(* PLC project Wiimote example, Beremiz Beremiz 1 *)
(* stored: creationDateTime 2012-09-12T23:30:19, modificationDateTime 2017-06-06T13:10:31 *)

PROGRAM main
  VAR
    x : INT;
    y : INT;
    a : INT;
    b : INT;
    c : INT;
    b1 : WORD;
    b0 : WORD;
  END_VAR
  VAR_EXTERNAL
    WiiNunchuckStickX : INT;
    WiiNunchuckStickY : INT;
    WiiNunchuckButtons : WORD;
    WiiButtons : WORD;
    WiiNunchuckAccX : INT;
    WiiNunchuckAccY : INT;
    WiiNunchuckAccZ : INT;
  END_VAR

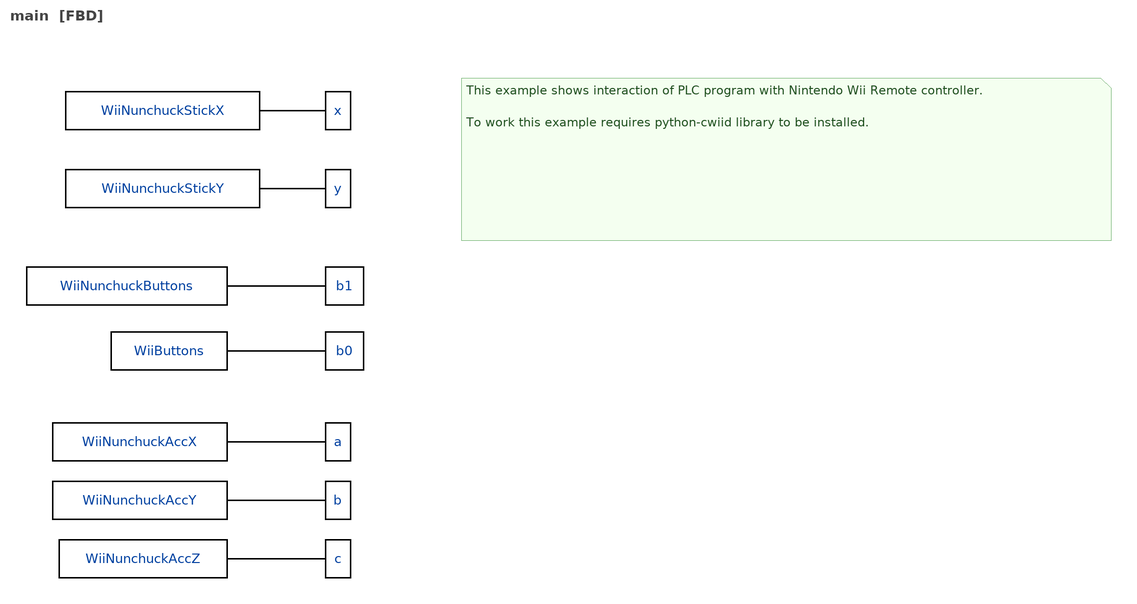
(* FBD diagram, written out as Structured Text *)
(* This example shows interaction of PLC program with Nintendo Wii Remote controller.

To work this example requires python-cwiid library to be installed. *)
x := WiiNunchuckStickX;
y := WiiNunchuckStickY;
b1 := WiiNunchuckButtons;
b0 := WiiButtons;
a := WiiNunchuckAccX;
b := WiiNunchuckAccY;
c := WiiNunchuckAccZ;
END_PROGRAM

CONFIGURATION config
  RESOURCE resource1 ON PLC
    TASK tsk1(INTERVAL := T#1ms, PRIORITY := 0);
    PROGRAM inst1 WITH tsk1 : main;
  END_RESOURCE
END_CONFIGURATION
